// TIA Portal V20 export
DATA_BLOCK "SP502"   // DB318
// stored: MemoryReserve 100
   VAR
      "UPPER 1-1 HEATER TEMPERATURE CONTROLLER ALARM" : Bool;
      SPARE : Bool;
      "UPPER 1-2 HEATER TEMPERATURE CONTROLLER ALARM" : Bool;
      SPARE_1 : Bool;
      "LOWER 1-1 HEATER TEMPERATURE CONTROLLER ALARM" : Bool;
      SPARE_2 : Bool;
      "LOWER 1-2 HEATER TEMPERATURE CONTROLLER ALARM" : Bool;
      SPARE_3 : Bool;
      "LOWER 1-3 HEATER TEMPERATURE CONTROLLER ALARM" : Bool;
      SPARE_4 : Bool;
      SPARE_5 : Bool;
      SPARE_6 : Bool;
      SPARE_7 : Bool;
      SPARE_8 : Bool;
      "VISION BUSY (STO)" : Bool;
      "VISION RESULT (OK)" : Bool;
   END_VAR
BEGIN
END_DATA_BLOCK
